{attribute 'GeneratedUsingTerminal: EL9930-0000-0017'}
{attribute addProperty BoxType "EL9930-0000-0017"}
{attribute addProperty Description "EL9930-0000, PROFIsafe-Segment-Abschlussklemme Primary"}
{attribute addProperty Physics "KKK"}
{attribute addProperty Id "IO_InputsEMPTY_STRUCTURE0IO_OutputsEMPTY_STRUCTURE0WcStateAT %I*WcState_9091E0EB2InfoDataAT %I*InfoData_32EB74EA10"}
{attribute addProperty CRC "3088473660"}
{attribute addProperty Size "12"}
TYPE EL9930_B8165E3C EXTENDS EtcSlaveTerminalBase_947E5A46 :
STRUCT
	{attribute addProperty Name "IO_Inputs"}
	IO_Inputs : EMPTY_STRUCTURE;
	{attribute addProperty Name "IO_Outputs"}
	IO_Outputs : EMPTY_STRUCTURE;
	{attribute addProperty Name "WcState"}
	WcState : WcState_9091E0EB;
	{attribute addProperty Name "InfoData"}
	InfoData : InfoData_32EB74EA;
END_STRUCT
END_TYPE

(* stored: Version 1.2.0.0, ProductVersion 3.1.4024.11
   DUT EL9930_B8165E3C: Id {ec6923ae-7eda-43e7-98fc-9e68b9ba5638} *)
